KUKA KRL data list: Station3.dat

&ACCESS RV
DEFDAT  Station3 PUBLIC

ENDDAT
